(* LS Electric XG5000 project: 신호등_프로젝트 *)
(* PLC LSPLC *)

PROGRAM 신호등 (* task: 스캔 프로그램 *)
VAR
    TENSEC : INT := 10;
    남은시간 AT %MW10 : INT;
    남은시간표시 : CTD_INT;
    보행대기 : TON;
    보행버튼 AT %MX0 : BOOL;
    보행신호 : BOOL;
    점등 : TON;
    점멸 : TON;
    제로 : INT := 0;
    중복신호방지 AT %MX6 : BOOL;
    차선_녹색램프 AT %MX1 : BOOL;
    차선_적색램프 AT %MX3 : BOOL;
    차선_황색램프 AT %MX2 : BOOL;
    차선_황적 : TON;
    카운터 : BOOL;
    횡단_녹색램프 AT %MX5 : BOOL;
    횡단_적색램프 AT %MX4 : BOOL;
    횡단_점등 : BOOL;
    횡단_점멸 : BOOL;
END_VAR
VAR
    _e1 : R_TRIG;
    _e2 : R_TRIG;
END_VAR

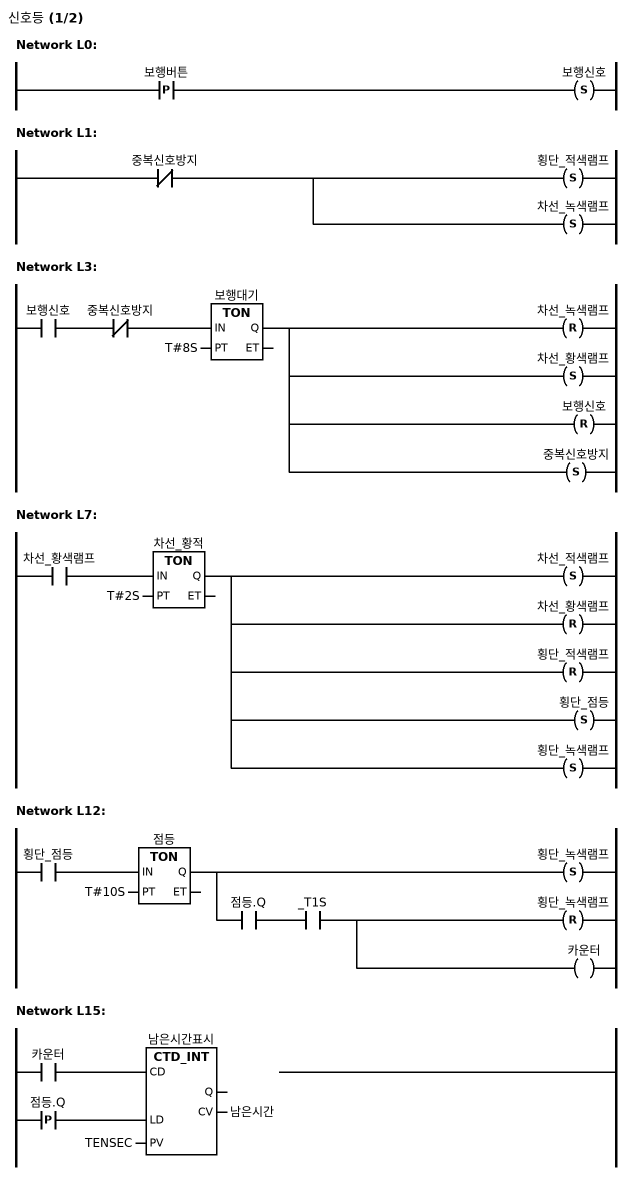
(* Rung L0 *)
_e1(CLK := 보행버튼);
IF _e1.Q THEN 보행신호 := TRUE; END_IF;
(* Rung L1 *)
IF NOT 중복신호방지 THEN
    횡단_적색램프 := TRUE;
    차선_녹색램프 := TRUE;
END_IF;
(* Rung L3 *)
보행대기(IN := 보행신호 AND NOT 중복신호방지, PT := T#8S);
IF 보행대기.Q THEN
    차선_녹색램프 := FALSE;
    차선_황색램프 := TRUE;
    보행신호 := FALSE;
    중복신호방지 := TRUE;
END_IF;
(* Rung L7 *)
차선_황적(IN := 차선_황색램프, PT := T#2S);
IF 차선_황적.Q THEN
    차선_적색램프 := TRUE;
    차선_황색램프 := FALSE;
    횡단_적색램프 := FALSE;
    횡단_점등 := TRUE;
    횡단_녹색램프 := TRUE;
END_IF;
(* Rung L12 *)
점등(IN := 횡단_점등, PT := T#10S);
IF 점등.Q THEN 횡단_녹색램프 := TRUE; END_IF;
IF 점등.Q AND 점등.Q AND _T1S THEN 횡단_녹색램프 := FALSE; END_IF;
카운터 := 점등.Q AND 점등.Q AND _T1S;
(* Rung L15 *)
_e2(CLK := 점등.Q);
남은시간표시(CD := 카운터, LD := _e2.Q, PV := TENSEC, CV => 남은시간);

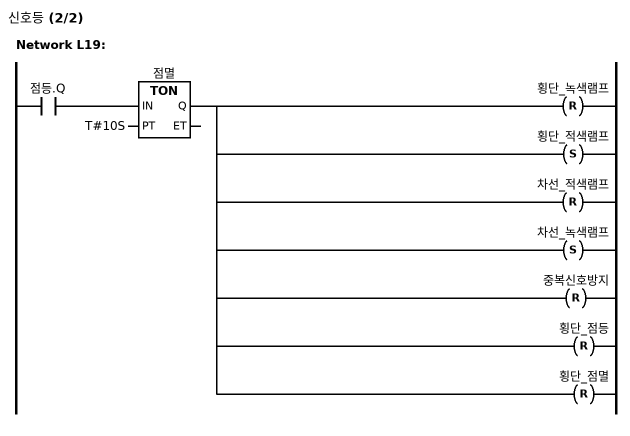
(* Rung L19 *)
점멸(IN := 점등.Q, PT := T#10S);
IF 점멸.Q THEN
    횡단_녹색램프 := FALSE;
    횡단_적색램프 := TRUE;
    차선_적색램프 := FALSE;
    차선_녹색램프 := TRUE;
    중복신호방지 := FALSE;
    횡단_점등 := FALSE;
    횡단_점멸 := FALSE;
END_IF;
END_PROGRAM